FUNCTION_BLOCK FB_Message EXTENDS FB_TcMessage
VAR_INPUT
	evtEntry	: TcEventEntry;
	bEvt		: BOOL;
END_VAR
VAR_OUTPUT
	bSent		: BOOL;
END_VAR
VAR
	rtrigSend	: R_TRIG;
	bInit	: BOOL := TRUE;
	bMem	: BOOL;
END_VAR

bSent := FALSE;
IF bInit THEN
	SUPER^.CreateEx(stEventEntry := evtEntry, ipSourceInfo := 0);
	bInit := FALSE;
END_IF

rtrigSend(CLK:= bEvt);
IF rtrigSend.Q THEN
	SUPER^.Send(0);
	bSent := TRUE;
END_IF

END_FUNCTION_BLOCK

(* stored: Version 1.1.0.1
   POU FB_Message: Id {072a73a1-3129-4aca-8d96-786d4205db36}, SpecialFunc None *)
